FUNCTION_BLOCK TEMPLATE_BASICFB
  (* Standard: 61499-2 *)
  (* Version 1.0, 11-01-12, GASR, Universidade do Estado de Santa Catarina *)
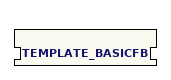
  EC_STATES
    START;
  END_STATES
END_FUNCTION_BLOCK
